FUNCTION_BLOCK ABSTRACT TcoCarouselBase EXTENDS TcoCore.TcoComponent

VAR_IN_OUT
	(*~
		<docu>
			<summary>
				In position sensor.
			</summary>	
		</docu>
	~*)
	inoInPosition : BOOL;
	(*~
		<docu>
			<summary>
				In precise position sensor.
			</summary>	
		</docu>
	~*)
	inoInPrecisePosition : BOOL;
END_VAR
VAR_IN_OUT
	(*~
		<docu>
			<summary>
				Enable turn signal.
			</summary>	
		</docu>
	~*)
	{attribute addProperty Name "<#Enable turn#>"}
	inoEnableTurn : BOOL;
	(*~
		<docu>
			<summary>
				Start turn  signal.
			</summary>	
		</docu>
	~*)
	{attribute addProperty Name "<#Start turn#>"}
	inoStartTurn : BOOL;
END_VAR
VAR

	{attribute addProperty Name "<#In position sensor#>"}
	_inPosition : BOOL;
	{attribute addProperty Name "<#In precise position sensor#>"}
	_inPrecisePosition : BOOL;
	(*~
		<docu>
			<summary>
				Enable turn  signal.
			</summary>	
		</docu>
	~*)
	{attribute addProperty Name "<#Enable turn table#>"}
	_enableTurn : BOOL;
	(*~
		<docu>
			<summary>
				Start trun signal.
			</summary>	
		</docu>
	~*)
	{attribute addProperty Name "<#Start turn table#>"}
	_startTurn : BOOL;
END_VAR

VAR
	{attribute addProperty Name "<#In position signal#>"}
	_InPositionSignalInfo : TcoCore.TcoSignalInfo;
	{attribute addProperty Name "<#In precise position signal#>"}
    _InPrecisePositionSignalInfo : TcoCore.TcoSignalInfo;
	{attribute addProperty Name "<#Enable turn signal#>"}
    _EnableTurnSignalInfo : TcoCore.TcoSignalInfo;
	{attribute addProperty Name "<#Start turn signal#>"}
    _StartTurnSignalInfo : TcoCore.TcoSignalInfo;
END_VAR

IF(__ISVALIDREF(inoInPosition)) THEN _inPosition := inoInPosition; _InPositionSignalInfo.GetSignalInfo(SIZEOF(inoInPosition), ADR(inoInPosition)); END_IF;
IF(__ISVALIDREF(inoInPrecisePosition)) THEN _inPrecisePosition := inoInPrecisePosition; _InPrecisePositionSignalInfo.GetSignalInfo(SIZEOF(inoInPrecisePosition), ADR(inoInPrecisePosition)); END_IF;
IF(__ISVALIDREF(inoEnableTurn)) THEN inoEnableTurn := _enableTurn; _EnableTurnSignalInfo.GetSignalInfo(SIZEOF(inoEnableTurn), ADR(inoEnableTurn)); END_IF;
IF(__ISVALIDREF(inoStartTurn)) THEN inoStartTurn := _startTurn; _StartTurnSignalInfo.GetSignalInfo(SIZEOF(inoStartTurn), ADR(inoStartTurn)); END_IF;

(*~
	<docu>
		<summary>
			Gets whether the carousel is in  position. 		
		</summary>			
	</docu>	
~*)
PROPERTY InPosition : bool
GET
InPosition := _inPosition;
END_GET
END_PROPERTY

(*~
	<docu>
		<summary>
			Gets whether the carousel is in precise position. 		
		</summary>			
	</docu>	
~*)
PROPERTY InPrecisePosition : bool
GET
InPrecisePosition := _inPrecisePosition;
END_GET
END_PROPERTY

(*~
	<docu>
		<summary>
			Restore all tasks of this instance into initial state.		 		 		
		</summary>			
	</docu>	
~*)
METHOD  Restore : ITcoRestorable
IF(TurnTask <> 0) THEN TurnTask.Restore(); END_IF;
END_METHOD

METHOD PROTECTED  ServiceMode
END_METHOD

(*~
	<docu>
		<summary>
			Starts rotating table. 		
		</summary>			
	</docu>	
~*)
METHOD Turn :TcoCore.ITcoTaskStatus
IF(TurnTask <> 0) THEN
	Turn := TurnTask.Invoke();
END_IF;
END_METHOD

(*~
	<docu>
		<summary>
			Starts rotating table do not check expected position 		
		</summary>			
	</docu>	
~*)
METHOD TurnRecovery :TcoCore.ITcoTaskStatus
IF(TurnTask <> 0) THEN

	TurnRecovery := TurnRecoveryTask.Invoke();
END_IF;
END_METHOD

(*~
	<docu>
		<summary>
			Gets the `TurnRecoveryTask` task that controls the rotation from  position to next position in same direction.
			<remarks>			
				<note type="important">
					This is an abstract method and must be implemented in derived class.
				</note>
			</remarks>	 		
		</summary>			
	</docu>	
~*)
PROPERTY PUBLIC ABSTRACT TurnRecoveryTask : TcoCore.ITcoTask
GET
END_GET
END_PROPERTY

(*~
	<docu>
		<summary>
			Gets the `TrunTask` task that controls the rotation from  position to next position in same direction.
			<remarks>			
				<note type="important">
					This is an abstract method and must be implemented in derived class.
				</note>
			</remarks>	 		
		</summary>			
	</docu>	
~*)
PROPERTY PUBLIC ABSTRACT TurnTask : TcoCore.ITcoTask
GET
END_GET
END_PROPERTY

END_FUNCTION_BLOCK

(* stored: Version 1.1.0.1, ProductVersion 3.1.4024.12
   POU TcoCarouselBase: Id {571c422a-c609-0b64-1fef-a02a776dca84}, SpecialFunc None
   Folder Operations: Id {3bae769a-4aca-0a30-1940-f1312a40fc2d}
   Folder States: Id {dfc95ad2-2cf9-032d-1a60-6015d0d43608}
   Folder Tasks: Id {2a40beee-6b4b-0667-29cc-3486b54c97cb}
   Property InPosition: Id {d69a896a-30ad-0e39-08ab-f27e02775f51}
   Get Get: Id {89e9d104-d929-0928-1826-6a474fa40668}
   Property InPrecisePosition: Id {8a98b7a0-30d2-09a8-009f-b8b23dc3285a}
   Get Get: Id {01253b06-3c1e-0c8a-13c7-a0ecc64d72e4}
   Method Restore: Id {368de314-cdb4-09a8-28ba-fffc6fc2c685}
   Method ServiceMode: Id {f4c3e8b5-c7e8-01f9-1196-a938272c1efc}
   Method Turn: Id {22e3e392-3f55-09ed-1c52-82d03f984974}
   Method TurnRecovery: Id {aba52f27-0f65-068c-13a7-8a141a19e8c9}
   Property TurnRecoveryTask: Id {59dbd72a-380a-06e5-2149-9fb319fb80e0}
   Get Get: Id {1471e626-b926-04be-0b68-4d0e211e11a5}
   Property TurnTask: Id {05f16e55-6df3-0265-3393-67ae5f28d889}
   Get Get: Id {12ccf9f1-5c36-0900-2e92-fa85e5dea42d} *)
